// TIA Portal project "PLCII_Pro10" (V15.1)

(* hardware
DEVICE "S7-1200 station_1"  S7-1200 Station
   slot 0: "Rack_0"  S7-1200 Rack  Rack  V1.0
   slot 1: "PLC_1"  CPU 1215C DC/DC/Rly  6ES7 215-1HG40-0XB0  V4.2
*)

// ===== PLC "PLC_1"  CPU 1215C DC/DC/Rly =====

VAR_GLOBAL   // PLC tag table "Default tag table"
   "Start" AT %M0.0 : Bool;
   "Sys_runing" AT %M0.1 : Bool;
   "Stop" AT %M0.2 : Bool;
   "Activate" AT %M0.3 : Bool;
   "Sys_Activated" AT %M0.4 : Bool;
END_VAR

DATA_BLOCK "SysVaribales"   // DB1
{ S7_Optimized_Access := 'TRUE' }
VERSION : 0.1
   VAR
      PB_Off : Bool;
      PB_Hand : Bool;
      PB_Auto : Bool;
      AutoCtrl : Bool;
      PumpMode : Int;
      PumpON : Bool;
      PumpOFF : Bool;
      All_AlarmInRst : Bool;
      Sys_cycleRunning : Bool;
      PumpStateInt : Int;
      FlowSW : Bool;
      PressureSn : Int;
      PressureRs : Real;
      FlowAlarm : Bool;
      FlowHorn : Bool;
      PressureAlarm : Bool;
      PressureHorn : Bool;
      AlarmReset : Bool;
      AlarmSilence : Bool;
      MaxPressure : Real;
   END_VAR
BEGIN
END_DATA_BLOCK

DATA_BLOCK "PumpControl_DB"   // DB2
{ S7_Optimized_Access := 'TRUE' }
VERSION : 0.1
// stored: InstanceOfName PumpControl
"PumpControl"
BEGIN
END_DATA_BLOCK

DATA_BLOCK "GettingPressure_DB"   // DB3
{ S7_Optimized_Access := 'TRUE' }
VERSION : 0.1
// stored: InstanceOfName GettingPressure
"GettingPressure"
BEGIN
END_DATA_BLOCK

FUNCTION_BLOCK "PumpControl"   // FB1, LAD
{ S7_Optimized_Access := 'TRUE' }
VERSION : 0.1
   VAR_INPUT
      Excute : Bool;
      PumpCycleTime : Time := T#7s;
      ResteCycleTime : Time := T#2s;
      PressureRS : Real := 30.0;
      MaxPressure : Real;
   END_VAR
   VAR
      HOA_Control_Instance_1 : "HOA_Control";
      IEC_Timer_0_Instance : TON_TIME;
      IEC_Timer_0_Instance_1 : TON_TIME;
      IEC_Timer_0_Instance_2 : TON_TIME;
      ons1 : Bool;
      ons2 : Bool;
      ons3 : Bool;
      ons4 : Bool;
      ons5 : Bool;
      ons6 : Bool;
      ons7 : Bool;
      IEC_Timer_0_Instance_3 : TON_TIME;
      PumpRunning : Bool;
      ons8 : Bool;
      Timer2 : Bool;
   END_VAR
   VAR CONSTANT
      Off_Mode : Int := 0;
      Hand_Mode : Int := 1;
      Auto_Mode : Int := 2;
   END_VAR
   VAR_TEMP   // added for the SCL form of the ladder/FBD networks
      _w1 : Bool;
      _w2 : Bool;
      _w3 : Bool;
   END_VAR
BEGIN

REGION Network 1
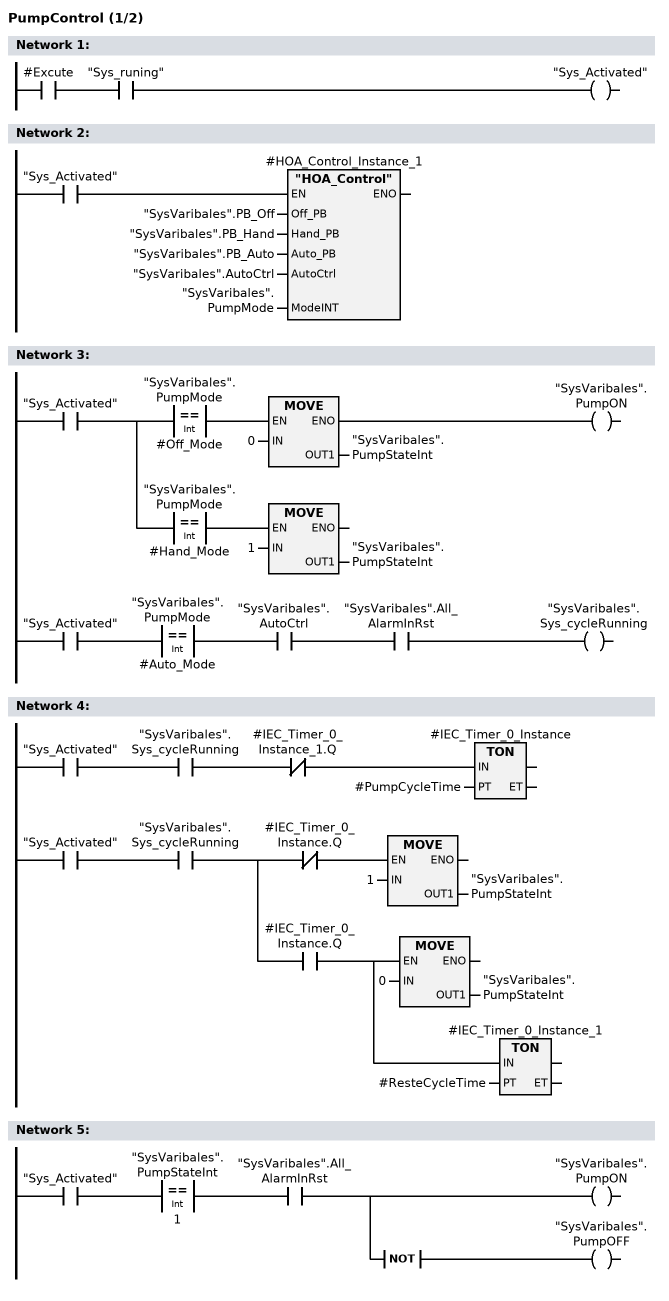
   RUNG wire#powerrail
      Contact( #Excute )
      Contact( "Sys_runing" )
      Coil( "Sys_Activated" )
   END_RUNG
   // the same network as SCL:
   "Sys_Activated" := #Excute AND "Sys_runing";
END_REGION

REGION Network 2
   RUNG wire#powerrail
      Contact( "Sys_Activated" )
      #HOA_Control_Instance_1(Off_PB := "SysVaribales".PB_Off, Hand_PB := "SysVaribales".PB_Hand, Auto_PB := "SysVaribales".PB_Auto, AutoCtrl := "SysVaribales".AutoCtrl, ModeINT := "SysVaribales".PumpMode)
   END_RUNG
   // the same network as SCL:
   IF "Sys_Activated" THEN
       #HOA_Control_Instance_1(Off_PB := "SysVaribales".PB_Off,   // "HOA_Control"
                               Hand_PB := "SysVaribales".PB_Hand,
                               Auto_PB := "SysVaribales".PB_Auto,
                               AutoCtrl := "SysVaribales".AutoCtrl,
                               ModeINT := "SysVaribales".PumpMode);
   END_IF;
END_REGION

REGION Network 3
   RUNG wire#powerrail
      Contact( "Sys_Activated" )
      wire#w1
      { S7_Templates := "SrcType := Int" } EQ_Contact(in1 := "SysVaribales".PumpMode, in2 := #Off_Mode)
      Move(in := 0, out1 => "SysVaribales".PumpStateInt)
      Coil( "SysVaribales".PumpON )
   END_RUNG
   RUNG wire#w1
      { S7_Templates := "SrcType := Int" } EQ_Contact(in1 := "SysVaribales".PumpMode, in2 := #Hand_Mode)
      Move(in := 1, out1 => "SysVaribales".PumpStateInt)
   END_RUNG
   RUNG wire#powerrail
      Contact( "Sys_Activated" )
      { S7_Templates := "SrcType := Int" } EQ_Contact(in1 := "SysVaribales".PumpMode, in2 := #Auto_Mode)
      Contact( "SysVaribales".AutoCtrl )
      Contact( "SysVaribales".All_AlarmInRst )
      Coil( "SysVaribales".Sys_cycleRunning )
   END_RUNG
   // the same network as SCL:
   #_w1 := "Sys_Activated" AND ("SysVaribales".PumpMode = #Off_Mode);
   IF #_w1 THEN "SysVaribales".PumpStateInt := 0; END_IF;
   "SysVaribales".PumpON := #_w1;
   IF "Sys_Activated" AND ("SysVaribales".PumpMode = #Hand_Mode) THEN
       "SysVaribales".PumpStateInt := 1;
   END_IF;
   "SysVaribales".Sys_cycleRunning := "Sys_Activated" AND ("SysVaribales".PumpMode = #Auto_Mode) AND "SysVaribales".AutoCtrl AND "SysVaribales".All_AlarmInRst;
END_REGION

REGION Network 4
   #IEC_Timer_0_Instance(IN := "Sys_Activated" AND "SysVaribales".Sys_cycleRunning AND NOT #IEC_Timer_0_Instance_1.Q,   // TON
                         PT := #PumpCycleTime);
   #_w1 := "Sys_Activated" AND "SysVaribales".Sys_cycleRunning;
   IF #_w1 AND NOT #IEC_Timer_0_Instance.Q THEN "SysVaribales".PumpStateInt := 1; END_IF;
   #_w2 := #_w1 AND #IEC_Timer_0_Instance.Q;
   IF #_w2 THEN "SysVaribales".PumpStateInt := 0; END_IF;
   #IEC_Timer_0_Instance_1(IN := #_w2, PT := #ResteCycleTime);   // TON
END_REGION

REGION Network 5
   RUNG wire#powerrail
      Contact( "Sys_Activated" )
      { S7_Templates := "SrcType := Int" } EQ_Contact(in1 := "SysVaribales".PumpStateInt, in2 := 1)
      Contact( "SysVaribales".All_AlarmInRst )
      wire#w1
      Coil( "SysVaribales".PumpON )
   END_RUNG
   RUNG wire#w1
      Not()
      Coil( "SysVaribales".PumpOFF )
   END_RUNG
   // the same network as SCL:
   "SysVaribales".PumpON := "Sys_Activated" AND ("SysVaribales".PumpStateInt = 1) AND "SysVaribales".All_AlarmInRst;
   "SysVaribales".PumpOFF := NOT "SysVaribales".PumpON;
END_REGION

REGION Network 6
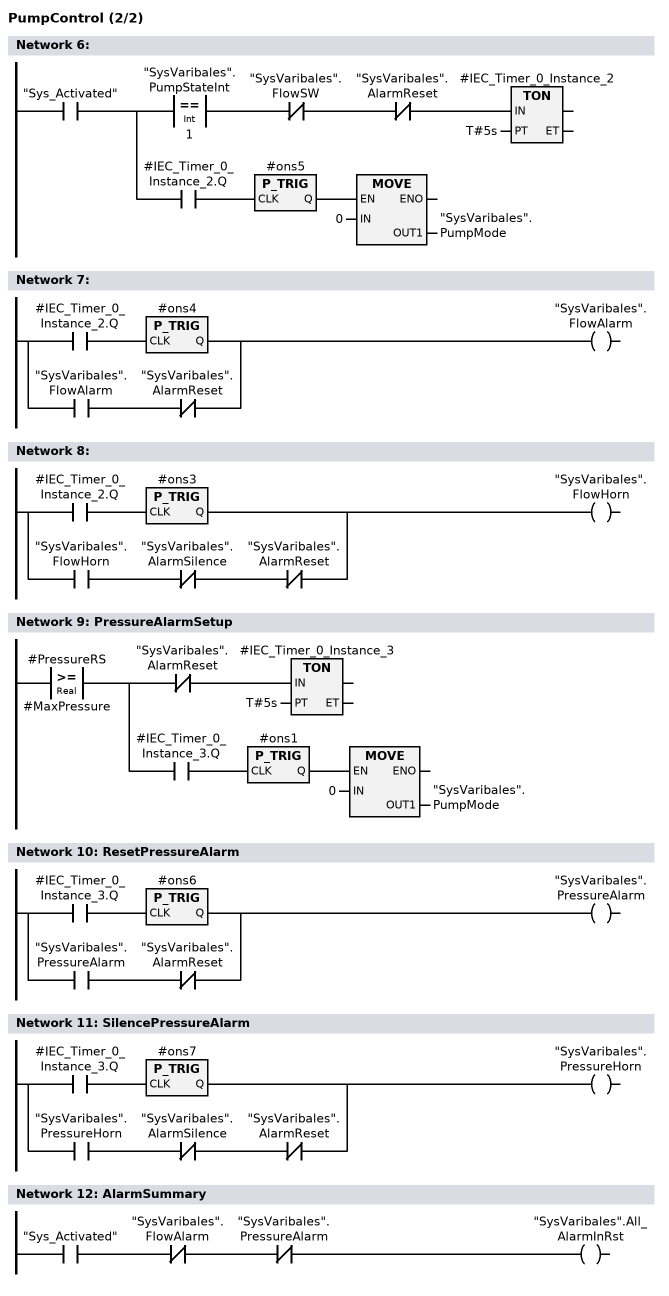
   #IEC_Timer_0_Instance_2(IN := "Sys_Activated" AND ("SysVaribales".PumpStateInt = 1) AND NOT "SysVaribales".FlowSW AND NOT "SysVaribales".AlarmReset,   // TON
                           PT := T#5s);
   #_w1 := "Sys_Activated" AND #IEC_Timer_0_Instance_2.Q;
   #_w2 := #_w1 AND NOT #ons5;   // rising edge
   #ons5 := #_w1;
   IF #_w2 THEN "SysVaribales".PumpMode := 0; END_IF;
END_REGION

REGION Network 7
   RUNG wire#powerrail
      Contact( #IEC_Timer_0_Instance_2.Q )
      P_Trig( #ons4 )
      wire#w1
      Coil( "SysVaribales".FlowAlarm )
   END_RUNG
   RUNG wire#powerrail
      Contact( "SysVaribales".FlowAlarm )
      I_Contact( "SysVaribales".AlarmReset )
   END_RUNG wire#w1
   // the same network as SCL:
   #_w1 := #IEC_Timer_0_Instance_2.Q AND NOT #ons4;   // rising edge
   #ons4 := #IEC_Timer_0_Instance_2.Q;
   "SysVaribales".FlowAlarm := #_w1 OR ("SysVaribales".FlowAlarm AND NOT "SysVaribales".AlarmReset);
END_REGION

REGION Network 8
   RUNG wire#powerrail
      Contact( #IEC_Timer_0_Instance_2.Q )
      P_Trig( #ons3 )
      wire#w1
      Coil( "SysVaribales".FlowHorn )
   END_RUNG
   RUNG wire#powerrail
      Contact( "SysVaribales".FlowHorn )
      I_Contact( "SysVaribales".AlarmSilence )
      I_Contact( "SysVaribales".AlarmReset )
   END_RUNG wire#w1
   // the same network as SCL:
   #_w1 := #IEC_Timer_0_Instance_2.Q AND NOT #ons3;   // rising edge
   #ons3 := #IEC_Timer_0_Instance_2.Q;
   "SysVaribales".FlowHorn := #_w1 OR ("SysVaribales".FlowHorn AND NOT "SysVaribales".AlarmSilence AND NOT "SysVaribales".AlarmReset);
END_REGION

REGION Network 9: PressureAlarmSetup
   #_w1 := #PressureRS >= #MaxPressure;
   #IEC_Timer_0_Instance_3(IN := #_w1 AND NOT "SysVaribales".AlarmReset, PT := T#5s);   // TON
   #_w2 := #_w1 AND #IEC_Timer_0_Instance_3.Q;
   #_w3 := #_w2 AND NOT #ons1;   // rising edge
   #ons1 := #_w2;
   IF #_w3 THEN "SysVaribales".PumpMode := 0; END_IF;
END_REGION

REGION Network 10: ResetPressureAlarm
   RUNG wire#powerrail
      Contact( #IEC_Timer_0_Instance_3.Q )
      P_Trig( #ons6 )
      wire#w1
      Coil( "SysVaribales".PressureAlarm )
   END_RUNG
   RUNG wire#powerrail
      Contact( "SysVaribales".PressureAlarm )
      I_Contact( "SysVaribales".AlarmReset )
   END_RUNG wire#w1
   // the same network as SCL:
   #_w1 := #IEC_Timer_0_Instance_3.Q AND NOT #ons6;   // rising edge
   #ons6 := #IEC_Timer_0_Instance_3.Q;
   "SysVaribales".PressureAlarm := #_w1 OR ("SysVaribales".PressureAlarm AND NOT "SysVaribales".AlarmReset);
END_REGION

REGION Network 11: SilencePressureAlarm
   RUNG wire#powerrail
      Contact( #IEC_Timer_0_Instance_3.Q )
      P_Trig( #ons7 )
      wire#w1
      Coil( "SysVaribales".PressureHorn )
   END_RUNG
   RUNG wire#powerrail
      Contact( "SysVaribales".PressureHorn )
      I_Contact( "SysVaribales".AlarmSilence )
      I_Contact( "SysVaribales".AlarmReset )
   END_RUNG wire#w1
   // the same network as SCL:
   #_w1 := #IEC_Timer_0_Instance_3.Q AND NOT #ons7;   // rising edge
   #ons7 := #IEC_Timer_0_Instance_3.Q;
   "SysVaribales".PressureHorn := #_w1 OR ("SysVaribales".PressureHorn AND NOT "SysVaribales".AlarmSilence AND NOT "SysVaribales".AlarmReset);
END_REGION

REGION Network 12: AlarmSummary
   RUNG wire#powerrail
      Contact( "Sys_Activated" )
      I_Contact( "SysVaribales".FlowAlarm )
      I_Contact( "SysVaribales".PressureAlarm )
      Coil( "SysVaribales".All_AlarmInRst )
   END_RUNG
   // the same network as SCL:
   "SysVaribales".All_AlarmInRst := "Sys_Activated" AND NOT "SysVaribales".FlowAlarm AND NOT "SysVaribales".PressureAlarm;
END_REGION
END_FUNCTION_BLOCK

FUNCTION_BLOCK "HOA_Control"   // FB2, LAD
{ S7_Optimized_Access := 'TRUE' }
VERSION : 0.1
   VAR_INPUT
      Off_PB : Bool;
      Hand_PB : Bool;
      Auto_PB : Bool;
      AutoCtrl : Bool;
   END_VAR
   VAR_IN_OUT
      ModeINT : Int;
   END_VAR
   VAR
      ons1 : Bool;
      ons2 : Bool;
      ons3 : Bool;
      ons4 : Bool;
      PreviosMode : Int;
   END_VAR
   VAR_TEMP   // added for the SCL form of the ladder/FBD networks
      _w1 : Bool;
      _w2 : Bool;
   END_VAR
BEGIN

REGION Network 1
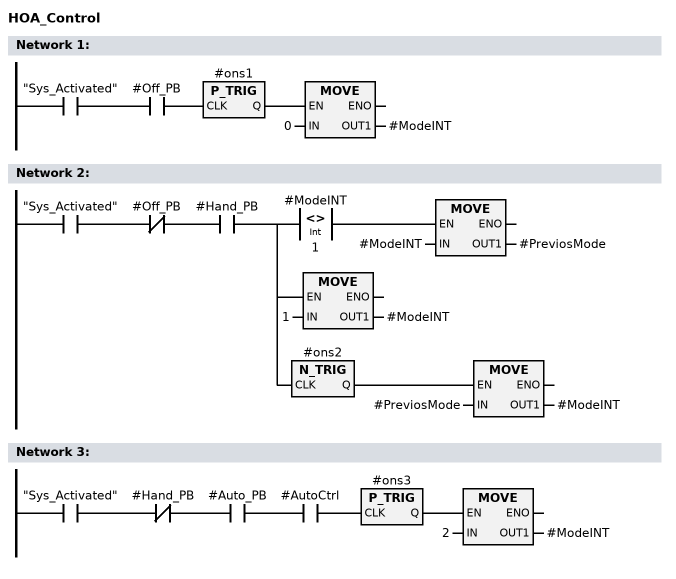
   RUNG wire#powerrail
      Contact( "Sys_Activated" )
      Contact( #Off_PB )
      P_Trig( #ons1 )
      Move(in := 0, out1 => #ModeINT)
   END_RUNG
   // the same network as SCL:
   #_w1 := "Sys_Activated" AND #Off_PB;
   #_w2 := #_w1 AND NOT #ons1;   // rising edge
   #ons1 := #_w1;
   IF #_w2 THEN #ModeINT := 0; END_IF;
END_REGION

REGION Network 2
   RUNG wire#powerrail
      Contact( "Sys_Activated" )
      I_Contact( #Off_PB )
      Contact( #Hand_PB )
      wire#w1
      { S7_Templates := "SrcType := Int" } NE_Contact(in1 := #ModeINT, in2 := 1)
      Move(in := #ModeINT, out1 => #PreviosMode)
   END_RUNG
   RUNG wire#w1
      Move(in := 1, out1 => #ModeINT)
   END_RUNG
   RUNG wire#w1
      N_Trig( #ons2 )
      Move(in := #PreviosMode, out1 => #ModeINT)
   END_RUNG
   // the same network as SCL:
   #_w1 := "Sys_Activated" AND NOT #Off_PB AND #Hand_PB;
   IF #_w1 AND (#ModeINT <> 1) THEN #PreviosMode := #ModeINT; END_IF;
   IF #_w1 THEN #ModeINT := 1; END_IF;
   #_w2 := NOT #_w1 AND #ons2;   // falling edge
   #ons2 := #_w1;
   IF #_w2 THEN #ModeINT := #PreviosMode; END_IF;
END_REGION

REGION Network 3
   RUNG wire#powerrail
      Contact( "Sys_Activated" )
      I_Contact( #Hand_PB )
      Contact( #Auto_PB )
      Contact( #AutoCtrl )
      P_Trig( #ons3 )
      Move(in := 2, out1 => #ModeINT)
   END_RUNG
   // the same network as SCL:
   #_w1 := "Sys_Activated" AND NOT #Hand_PB AND #Auto_PB AND #AutoCtrl;
   #_w2 := #_w1 AND NOT #ons3;   // rising edge
   #ons3 := #_w1;
   IF #_w2 THEN #ModeINT := 2; END_IF;
END_REGION
END_FUNCTION_BLOCK

FUNCTION_BLOCK "GettingPressure"   // FB3, LAD
{ S7_Optimized_Access := 'TRUE' }
VERSION : 0.1
   VAR_INPUT
      MinPr : Int;
      MaxPr : Int;
      PressureMesured : Int;
   END_VAR
   VAR_OUTPUT
      PressureResultedREAL : Real;
   END_VAR
   VAR_TEMP
      PrTemp : Real;
      PressureResultedINT : Real;
   END_VAR
BEGIN

REGION Network 1
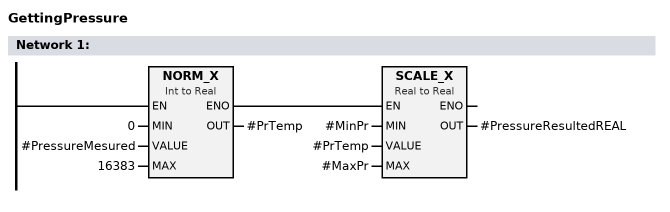
   RUNG wire#powerrail
      { S7_Templates := "[SrcType := Int, DestType := Real]" } Normalize(min := 0, value := #PressureMesured, max := 16383, out => #PrTemp)
      { S7_Templates := "[SrcType := Real, DestType := Real]" } Scale(min := #MinPr, value := #PrTemp, max := #MaxPr, out => #PressureResultedREAL)
   END_RUNG
   // the same network as SCL:
   #PrTemp := NORM_X(MIN := 0, VALUE := #PressureMesured, MAX := 16383);
   #PressureResultedREAL := SCALE_X(MIN := #MinPr, VALUE := #PrTemp, MAX := #MaxPr);
END_REGION
END_FUNCTION_BLOCK

ORGANIZATION_BLOCK "Main"   // OB1, LAD, ProgramCycle
TITLE = "Main Program Sweep (Cycle)"
{ S7_Optimized_Access := 'TRUE' }
VERSION : 0.1
   VAR_INPUT
      Initial_Call : Bool;   // Initial call of this OB
      Remanence : Bool;   // =True, if remanent data are available
   END_VAR
BEGIN

REGION Network 1
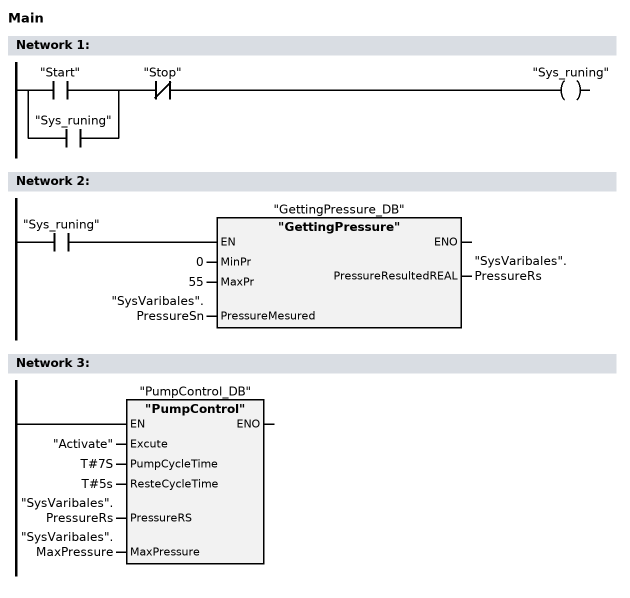
   RUNG wire#powerrail
      Contact( "Start" )
      wire#w1
      I_Contact( "Stop" )
      Coil( "Sys_runing" )
   END_RUNG
   RUNG wire#powerrail
      Contact( "Sys_runing" )
   END_RUNG wire#w1
   // the same network as SCL:
   "Sys_runing" := ("Start" OR "Sys_runing") AND NOT "Stop";
END_REGION

REGION Network 2
   RUNG wire#powerrail
      Contact( "Sys_runing" )
      "GettingPressure_DB"(MinPr := 0, MaxPr := 55, PressureMesured := "SysVaribales".PressureSn, PressureResultedREAL => "SysVaribales".PressureRs)
   END_RUNG
   // the same network as SCL:
   IF "Sys_runing" THEN
       "GettingPressure_DB"(MinPr := 0,   // "GettingPressure"
                            MaxPr := 55,
                            PressureMesured := "SysVaribales".PressureSn,
                            PressureResultedREAL => "SysVaribales".PressureRs);
   END_IF;
END_REGION

REGION Network 3
   RUNG wire#powerrail
      "PumpControl_DB"(Excute := "Activate", PumpCycleTime := T#7S, ResteCycleTime := T#5s, PressureRS := "SysVaribales".PressureRs, MaxPressure := "SysVaribales".MaxPressure)
   END_RUNG
   // the same network as SCL:
   "PumpControl_DB"(Excute := "Activate",   // "PumpControl"
                    PumpCycleTime := T#7S,
                    ResteCycleTime := T#5s,
                    PressureRS := "SysVaribales".PressureRs,
                    MaxPressure := "SysVaribales".MaxPressure);
END_REGION
END_ORGANIZATION_BLOCK